TYPE ST_BaseComplexElement_HMI :
STRUCT
END_STRUCT
END_TYPE

(* stored: Version 1.1.0.1
   DUT ST_BaseComplexElement_HMI: Id {ae2a4ff4-1f22-0aec-2d02-3ad5742d139e} *)
